FUNCTION F_Concat3 : T_MaxString
VAR_INPUT
   StringOne : STRING;
   StringTwo : STRING;
   StringThree : STRING;
END_VAR
VAR
   response : T_MaxString;
END_VAR

response := CONCAT(StringOne, StringTwo);
response := CONCAT(response, StringThree);
F_Concat3 := response;

END_FUNCTION

(* stored: Version 1.1.0.1, ProductVersion 3.1.4026.12
   POU F_Concat3: Id {9cf63a97-c84e-0f0d-1ab3-ca1e631333e8}, SpecialFunc None *)
